// TIA Portal V16 export
// export: Created 2021-11-12T13:33:11.8380753Z, ExportSetting WithDefaults, DisplayName Totally Integrated Automation Portal, DisplayVersion V16 Update 3, DisplayName TIA Portal Version Control Interface, DisplayVersion V16 Update 2, DisplayName TIA Portal Openness, DisplayVersion V16 Update 3, DisplayName SINAMICS Startdrive Advanced, DisplayVersion V16 Update 5, DisplayName SINAMICS Startdrive G130, G150, S120, S150, SINAMICS MV, S210, DisplayVersion V16 Update 5, DisplayName SINAMICS Startdrive G110M, G120, G120C, G120D, G120P, G115D, DisplayVersion V16 Update 5, DisplayName STEP 7 Professional, DisplayVersion V16 Update 3, DisplayName STEP 7 Safety, DisplayVersion V16, DisplayName WinCC UA Professional, DisplayVersion V16 Update 3
DATA_BLOCK "STD_Station_DB"   // DB222
{ DB_Accessible_From_OPC_UA := 'FALSE' }
VERSION : 0.1
// stored: AutoNumber true, DBAccessibleFromOPCUA false, InstanceOfName STD_Station, InstanceOfType FB
"STD_Station"
   // VAR_INPUT
   //    IS_ZoneM : "UDT_Status_main";
   //    IS_ZoneS : "UDT_Zone_Status_specific";
   //    IB1StnExtCtrl : Bool;
   //    IB1StnAutoRun : Bool;
   //    IB1Rmt : Bool;
   //    IB1ManSwch : Bool;
   //    IB1AutSwch : Bool;
   //    IB1SftyOK : Bool;
   //    IB1Run : Bool;
   //    IB1CollWrn : Bool;
   //    IB1CollErr : Bool;
   //    IB1AllAutoRun : Bool;
   //    IB1AllEndOfCycle : Bool;
   //    IB1AllEndOfProd : Bool;
   //    IB1AllInBasePos : Bool;
   //    IB1AllStopBefor : Bool;
   //    IB1AllStopAfter : Bool;
   //    IB1ReqBasePos : Bool;
   //    IB1ReqEndOfCycle : Bool;
   //    IB1ReqEndOfProdAct : Bool;
   //    IB1ReqEndOfProdCncl : Bool;
   //    IB1AutStartBtn : Bool;
   //    IB1Stop : Bool;
   //    IB1Blink : Bool;
   //    IB1AlmSupp : Bool;
   //    II_DevSelNr : Int;
   // END_VAR
   // VAR_OUTPUT
   //    OS_Status : Struct
   //       Main : "UDT_Status_main";
   //       Specific : "UDT_Zone_Status_specific";
   //       Error : "UDT_Error01";
   //    END_STRUCT;
   //    OB1AutStart : Bool;
   //    OB1Man : Bool;
   //    OB1Rmt : Bool;
   //    OB1SigAcs : Bool;
   // END_VAR
   // VAR_IN_OUT
   //    XS_Parameter : "UDT_Station_Parameter";
   //    XS_Command : "UDT_Station_Command";
   // END_VAR
   // VAR
   //    SS_Alarm : Struct
   //       Res_0_0 : Bool;
   //       Res_0_1 : Bool;
   //       Res_0_2 : Bool;
   //       Res_0_3 : Bool;
   //       Res_0_4 : Bool;
   //       Res_0_5 : Bool;
   //       Res_0_6 : Bool;
   //       Res_0_7 : Bool;
   //    END_STRUCT;
   //    SS_Warning : Struct
   //       EndOfCycle : Bool;
   //       EndOfProd : Bool;
   //       StepMode : Bool;
   //       StopBefor : Bool;
   //       StopAfter : Bool;
   //       BypasMode : Bool;
   //       Res_0_6 : Bool;
   //       Res_0_7 : Bool;
   //    END_STRUCT;
   //    SB1AutoRun : Bool;
   //    SB1AutoRunBasePos : Bool;
   //    SB1AutoRunProd : Bool;
   //    SB1ModeAutStep : Bool;
   //    SB1ModeStopBefor : Bool;
   //    SB1ModeStopAfter : Bool;
   //    SB1ModeBypas : Bool;
   //    SB1ModeAut : Bool;
   //    SB1ModeMan : Bool;
   //    SB1ModeOff : Bool;
   //    SB1ReqEndOfCycle : Bool;
   //    SB1ReqEndOfProd : Bool;
   //    SB1ManAutPE : Bool;
   //    SB1OffPE : Bool;
   //    SB1ReqBasePosPE : Bool;
   //    SB1ReqEndOfCyclePE : Bool;
   //    SB1ReqEndOfProdActPE : Bool;
   //    SB1ReqEndOfProdCnclPE : Bool;
   //    SB1AutStart : Bool;
   //    SB1AutStartAux : Bool;
   //    SB1AuxHorn : Bool;
   //    SB1AutStartBtnPE : Bool;
   //    ST_Horn { S7_SetPoint := 'True'} : TON_TIME;
   //    ST_Start { S7_SetPoint := 'True'} : TON_TIME;
   //    ST_AlmSupp { S7_SetPoint := 'True'} : IEC_TIMER;
   // END_VAR
BEGIN
END_DATA_BLOCK
